(* IEC 61131-3 sources: AXOpen/src/core/ctrl/src/AxoDialog, 8 files *)

(* ---- eDialogAnswer.st ---- *)
NAMESPACE AXOpen.Core
    TYPE
        eDialogAnswer : INT (
            NoAnswer := 0,
            OK := 10,
            Yes := 20,
            No := 30,
            Cancel := 40
        );
    END_TYPE
END_NAMESPACE

(* ---- eDialogButtons.st ---- *)
NAMESPACE AXOpen.Core
    TYPE
        eDialogButtons : INT (
            NoButtons := 0,
            Ok := 10,
            YesNo := 20,
            YesNoCancel := 30
        );
    END_TYPE
END_NAMESPACE

(* ---- eDialogType.st ---- *)
NAMESPACE AXOpen.Core
    TYPE
        eDialogType : INT (
            Undefined := 0,
            Info := 10,
            Success := 20,
            Danger := 30,
            Warning := 40
        );
    END_TYPE
END_NAMESPACE

(* ---- IAxoDialogAnswer.st ---- *)
NAMESPACE AXOpen.Core
    INTERFACE IAxoDialogAnswer EXTENDS IAxoDialogFormat

        METHOD Answer : eDialogAnswer
        END_METHOD

    END_INTERFACE
END_NAMESPACE

(* ---- IAxoDialogFormat.st ---- *)
NAMESPACE AXOpen.Core
    INTERFACE PUBLIC IAxoDialogFormat
        METHOD WithCaption : IAxoDialogAnswer
            VAR_INPUT
                inCaption : STRING;
            END_VAR
        END_METHOD

        METHOD WithOk : IAxoDialogAnswer
        END_METHOD

        METHOD WithText : IAxoDialogAnswer
            VAR_INPUT
                inText : STRING;
            END_VAR
        END_METHOD

        METHOD WithType : IAxoDialogAnswer
            VAR_INPUT
                inDialogType : eDialogType;
            END_VAR
        END_METHOD

        METHOD WithYesNo : IAxoDialogAnswer
        END_METHOD

        METHOD WithYesNoCancel : IAxoDialogAnswer
        END_METHOD
    END_INTERFACE
END_NAMESPACE

(* ---- AxoAlertDialog.st ---- *)
NAMESPACE AXOpen.Core
    CLASS PUBLIC AxoAlertDialog EXTENDS AxoDialogBase

        VAR PUBLIC
            _dialogType : eDialogType;
            _title : STRING;
            _message : STRING;
            _timeToBurn : INT;
        END_VAR

        METHOD PUBLIC Show : IAxoTaskState
            VAR_INPUT
                _parent : IAxoObject;
                DialogType : eDialogType;
                Title : STRING;
                Message : STRING;
                TimeToBurn : INT;
            END_VAR

            THIS.Initialize(_parent);

            Show := THIS.Invoke();
            SUPER.Execute();

            _dialogType := DialogType;
            _title := Title;
            _message := Message;
            _timeToBurn := TimeToBurn;
        END_METHOD

END_CLASS
END_NAMESPACE

(* ---- AxoDialog.st ---- *)
NAMESPACE AXOpen.Core
    ///<summary>
    /// AxoDialog class, which represents structure of base dialog.
    ///</summary>
    {S7.extern=ReadWrite}
    CLASS PUBLIC AxoDialog EXTENDS AxoDialogBase IMPLEMENTS IAxoDialogFormat, IAxoDialogAnswer

        VAR PUBLIC
            _text : STRING;
            _caption : STRING;
            _buttons : eDialogButtons;
            _answer : eDialogAnswer;
            _dialogType : eDialogType;
        END_VAR

        VAR PRIVATE
            _risingEdge : BOOL;  // not used in .net side
            _lastCall : ULINT;
            _createPlcCycleSpace :  BOOL;
            _PlcCycleSpaceCounter : UINT;
        END_VAR

        ///<summary>
        /// Show method, which serves for initializing remote task and invoking dialog from PLC.
        ///</summary>
        METHOD PUBLIC Show : IAxoDialogFormat
            VAR_INPUT
                inParent : IAxoObject;
            END_VAR

            VAR_TEMP
                callCounter : ULINT;
            END_VAR

            SUPER.SuspendExecuteAnalisis();

            Show := THIS;

            IF(inParent = NULL) THEN RETURN; END_IF;

            SUPER.Run(inParent);

            IF NOT THIS.IsInitialized THEN // dialog is not observed/monitored by server

                IF (THIS.Status <> eAxoTaskState#Ready) THEN
                    THIS.Restore();
                end_if;

                _answer := eDialogAnswer#NoAnswer; // set default value
                ErrorDetails := 'THE REMOTE TASK IS NOT INITIALIZED';
                RETURN; // if it continue  .Execute() call ThrowWhen() and task go to ErrorState
            END_IF;

            callCounter := THIS.GetParent().GetContext().OpenCycleCount();
            if callCounter = _lastCall then //is called in the same cycle, suppose that is a new dialog
                _answer := eDialogAnswer#NoAnswer; // must be reseted.
                RETURN;
            END_IF;

            IF _createPlcCycleSpace THEN // create cycle space AFTER RESPONSE
                _answer := eDialogAnswer#NoAnswer; // must be set due to call for new dialog.
                _PlcCycleSpaceCounter  := _PlcCycleSpaceCounter + UINT#1;
                IF _PlcCycleSpaceCounter > UINT#2 then // IT IS REDUNDAND
                    _createPlcCycleSpace := FALSE;
                END_IF;
                RETURN;
            END_IF;

            // Restores when not called for 2+ consecutive cycles of the context.
            IF(callCounter > _lastCall + ULINT#1) THEN
                THIS.Restore();
                _answer := eDialogAnswer#NoAnswer;
            END_IF;
            _lastCall := callCounter;

            IF (THIS.Status = eAxoTaskState#Ready) THEN
                _closeSignal := FALSE;
            END_IF;

            THIS.Invoke();
            SUPER.Execute();

            //after task is done and some answer is provided, restore this task
            IF (THIS.Status = eAxoTaskState#Done && _answer <> eDialogAnswer#NoAnswer) THEN
                THIS.Restore();
                _createPlcCycleSpace := true;
            END_IF;
         END_METHOD

        ///<summary>
        /// Show method with a possibility to close dialog externally by setting a signal.
        /// WARNING: This is experimental implementation of possibility to close dialogs externally. More testing need to be done.
        ///</summary>
        METHOD PUBLIC ShowWithExternalClose : IAxoDialogFormat
            VAR_INPUT
                inParent : IAxoObject;
                inOkAnswerSignal : BOOL := FALSE;
                inYesAnswerSignal : BOOL := FALSE;
                inNoAnswerSignal : BOOL := FALSE;
                inCancelAnswerSignal : BOOL := FALSE;
            END_VAR

            VAR_TEMP
                callCounter : ULINT;
                edgeDetected : BOOL;
            END_VAR

            ShowWithExternalClose := THIS;

            IF(inParent = NULL) THEN
                RETURN;
            END_IF;

            SUPER.Run(inParent);

            IF NOT THIS.IsInitialized THEN // dialog is not observed/monitored by server
                _answer := eDialogAnswer#NoAnswer; // set default value
                ErrorDetails := 'THE REMOTE TASK IS NOT INITIALIZED';
                RETURN; // if it continue  .Execute() call ThrowWhen() and task go to ErrorState
            END_IF;

            callCounter := THIS.GetParent().GetContext().OpenCycleCount();
            if callCounter = _lastCall then //is called in the same cycle, suppose that is a new dialog
                _answer := eDialogAnswer#NoAnswer; // must be reseted.
                RETURN;
            END_IF;

            IF _createPlcCycleSpace THEN // create cycle space AFTER RESPONSE
                _answer := eDialogAnswer#NoAnswer; // must be set due to call for new dialog.
                _PlcCycleSpaceCounter  := _PlcCycleSpaceCounter + UINT#1;
                IF _PlcCycleSpaceCounter > UINT#2 then // IT IS REDUNDAND
                    _createPlcCycleSpace := FALSE;
                    _PlcCycleSpaceCounter:=  UINT#0;
                END_IF;
                RETURN;
            END_IF;

            // Restores when not called for 2+ consecutive cycles of the context.
            IF(callCounter > _lastCall + ULINT#1) THEN
                THIS.Restore();
                _answer := eDialogAnswer#NoAnswer;
            END_IF;
            _lastCall := callCounter;

            IF (THIS.Status = eAxoTaskState#Ready) THEN
                _closeSignal := FALSE;
            END_IF;

            THIS.Invoke();
            SUPER.Execute();

            // watch close signals on rising edge
            edgeDetected := ((inOkAnswerSignal XOR inYesAnswerSignal XOR inNoAnswerSignal XOR inCancelAnswerSignal) AND NOT _risingEdge);
            _risingEdge := inOkAnswerSignal XOR inYesAnswerSignal XOR inNoAnswerSignal XOR inCancelAnswerSignal;

            IF edgeDetected THEN
                _closeSignal := TRUE;
                IF inOkAnswerSignal THEN
                    _answer := eDialogAnswer#Ok;
                ELSIF	inYesAnswerSignal THEN
                    _answer := eDialogAnswer#Yes;
                ELSIF	inNoAnswerSignal THEN
                    _answer := eDialogAnswer#No;
                ELSIF	inCancelAnswerSignal THEN
                    _answer := eDialogAnswer#Cancel;
                END_IF;

            END_IF;

            //after task is done and some answer is provided, restore this task
            IF (THIS.Status = eAxoTaskState#Done && _answer <> eDialogAnswer#NoAnswer) THEN
                THIS.Restore();
                _createPlcCycleSpace := true;
            END_IF;

        END_METHOD

        ///<summary>
        /// Executes once when the task is restored.
        ///</summary>
        METHOD PROTECTED OVERRIDE OnRestore
            SUPER.OnRestore();
            _buttons := eDialogButtons#NoButtons;
            _text := '';
            _caption := '';
            _dialogType := eDialogType#Undefined;

            _createPlcCycleSpace :=  FALSE;
            _PlcCycleSpaceCounter:=  UINT#0;
        END_METHOD

    METHOD PUBLIC WithCaption : IAxoDialogAnswer
        VAR_INPUT
            inCaption : STRING;
        END_VAR

        _caption := inCaption;
        WithCaption := THIS;
    END_METHOD

    METHOD PUBLIC WithOk : IAxoDialogAnswer
        _buttons := eDialogButtons#Ok;
        WithOk := THIS;
    END_METHOD

    METHOD PUBLIC WithText : IAxoDialogAnswer
        VAR_INPUT
            inText : STRING;
        END_VAR

        _text := inText;
        WithText := THIS;
    END_METHOD

    METHOD PUBLIC WithType : IAxoDialogAnswer
        VAR_INPUT
            inDialogType : eDialogType;
        END_VAR

        _dialogType := inDialogType;
        WithType := THIS;
    END_METHOD

    METHOD PUBLIC WithYesNo : IAxoDialogAnswer
        _buttons := eDialogButtons#YesNo;
        WithYesNo := THIS;
    END_METHOD

    METHOD PUBLIC WithYesNoCancel : IAxoDialogAnswer
        _buttons := eDialogButtons#YesNoCancel;
        WithYesNoCancel := THIS;
    END_METHOD

    METHOD PUBLIC Answer : eDialogAnswer
        Answer := _answer;
    END_METHOD

END_CLASS
END_NAMESPACE

(* ---- AxoDialogBase.st ---- *)
NAMESPACE AXOpen.Core
    {S7.extern=ReadWrite}
    CLASS PUBLIC AxoDialogBase EXTENDS AxoRemoteTask
        VAR PUBLIC
            _closeSignal : BOOL;
        END_VAR

        ///<summary>
        /// Restore dialog. In special case context can be null.
        ///</summary>
        METHOD PUBLIC OVERRIDE Restore : IAxoTaskState
            Restore := THIS;

            IF _context = NULL THEN
                Status := eAxoTaskState#Ready;  //needed in case when dialog observation was interrupt
                ErrorDetails := '';
                THIS.OnRestore();
            ELSE
                SUPER.Restore();
            END_IF;
        END_METHOD

        ///<summary>
        /// Executes once when the task is restored.
        ///</summary>
        METHOD PROTECTED OVERRIDE OnRestore
            _closeSignal := true; // close all dialogs...
        END_METHOD
    END_CLASS
END_NAMESPACE
